// Gets the upper bound index of the array of specified type.
FUNCTION F_GetXWordArrayUpperBound : T_Position // The upper bound index of the specified array.
VAR_IN_OUT
	arArray : ARRAY[*] OF __XWORD; // The array to query.
END_VAR

F_GetXWordArrayUpperBound := UPPER_BOUND(arArray, 1);

END_FUNCTION

(* stored: Version 1.1.0.1
   POU F_GetXWordArrayUpperBound: Id {c1f98c39-1b85-0543-0b77-bac626047c95}, SpecialFunc None *)
